Fanuc KAREL source: untitled1.kl

%NOLOCKGROUP
%COMMENT = 'RESUME ROS TASKS'

PROGRAM ros_resume
BEGIN
end ros_resume
